Staubli VAL3: getDefaultType.pgx

public program getDefaultType(num& x_nType[])
begin
  // get the process List
  // get the last type used
  x_nType=saveCycle:nType
end
